FUNCTION_BLOCK BasicCalcEmpty (* Basic FB with empty ECC *)
  (* Standard: 61499-2 *)
  (* Version 1.0, 2023-07-26, AK115394 *)
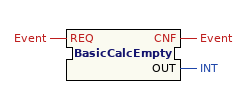
  EVENT_INPUT
    REQ;
  END_EVENT
  EVENT_OUTPUT
    CNF;
  END_EVENT
  VAR_OUTPUT
    OUT : INT;
  END_VAR
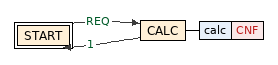
  EC_STATES
    START; (* Initial State *)
    CALC : calc -> CNF;
  END_STATES
  EC_TRANSITIONS
    START TO CALC := REQ;
    CALC TO START := 1;
  END_TRANSITIONS
  ALGORITHM calc IN ST:
	OUT:=1;
  END_ALGORITHM
END_FUNCTION_BLOCK
